Fanuc KAREL source: kt00567.KL

-- PROVISIONAL review KL for V940-1; original PC SHA256 44f1dac464e636130c4ef129a56706116bbf06e0a4ca572f46f5330c698f4655
-- Incomplete behavior may be omitted. Consult companion uncertainty JSON. Do not deploy.
PROGRAM KT00567
%NOLOCKGROUP
VAR
  R2 : REAL
-- UNRESOLVED_DECL V1 type=000013
-- UNRESOLVED_DECL OUT type=000013
BEGIN
  -- V9_ZERO_TABLE_METADATA_HINT layout=0001; no indexed target words; source/name/runtime held
  -- UNRESOLVED_PC offsets 5-20; opcodes 2E,22,32,35
  -- UNRESOLVED_PC offsets 25-36; opcodes 2E,23
  -- UNRESOLVED_PC offsets 41-63; opcodes 49,21,8A,4A
  -- UNRESOLVED_PC offsets 68-72; opcodes 7F
END KT00567
